(*
SPDX-FileCopyrightText: Â© 2026 Oleksandr Tiutyk <trofimich@gmail.com>
SPDX-License-Identifier: MIT
License: https://opensource.org/license/mit
*)

(*!
<summary>Provides cyclic execution and initialization state of automation components.</summary>
<description>
Execute advances the fixed sequence of roots bound at construction. State and StateName describe runner initialization.
</description>
*)

INTERFACE IAutomationRunner EXTENDS TOF_Core.IObject

(*!
<summary>Initializes and advances cyclic execution of the registered components.</summary>
<description>
Validates the bound roots before the first root initialization. An empty array, null slot or repeated instance
makes the runner INVALID. After initialization succeeds, subsequent calls execute roots in array order.
Call from the outer task boundary. Nested runner execution is unsupported because cleanup covers the calling task.
Call at the task boundary outside handlers that swallow terminal allocation failures.
</description>
*)
METHOD FINAL Execute
END_METHOD

(*!
<summary>Gets current initialization and operational state of the runner.</summary>
*)
{attribute 'monitoring' := 'call'}
PROPERTY FINAL State : AUTOMATION_RUNNER_STATE
GET
END_GET
END_PROPERTY

(*!
<summary>Gets string representation of current runner state.</summary>
*)
{attribute 'monitoring' := 'call'}
PROPERTY StateName : STRING
GET
END_GET
END_PROPERTY

END_INTERFACE

(* stored: Version 1.1.0.1
   Itf IAutomationRunner: Id {f1f89d3f-0708-4d4a-a276-5286e009b7ba}
   Method Execute: Id {43b25f17-24a8-4738-8b58-a34b4ca8299e}
   Property State: Id {67795c22-5567-4678-a754-1c0f3c5ade49}
   Get Get: Id {fb95b05a-71ee-4fbb-b12d-3b4b27b06a7a}
   Property StateName: Id {c3740711-6982-474a-957a-4fff61ca98ad}
   Get Get: Id {457a8b5e-1646-48ee-9ef4-f8250d06162a} *)
